// TIA Portal V21 export
DATA_BLOCK "FB_Write_Value_To_Word_DB"   // DB24
AUTHOR : JEBU
FAMILY : VTEMdc
VERSION : 1.0
// stored: InstanceOfName FB_Write_Value_To_Word, InstanceOfType FB
"FB_Write_Value_To_Word"
   // VAR_INPUT
   //    iValue { ExternalVisible := 'False'} : Int := 0;
   //    iStartBit { ExternalVisible := 'False'} : Int := 0;
   //    iEndBit { ExternalVisible := 'False'} : Int := 15;
   // END_VAR
   // VAR_OUTPUT
   //    xError { ExternalVisible := 'False'} : Bool := FALSE;
   // END_VAR
   // VAR_IN_OUT
   //    wDataWord { ExternalVisible := 'False'} : Word := 16#0000;
   // END_VAR
   // VAR
   //    wData { ExternalVisible := 'False'} : Word := 16#0000;
   // END_VAR
BEGIN
END_DATA_BLOCK
